(* IEC 61131-3 sources: NachHouse_CORE/V200/APP (part 6) *)

              47 : // HEV
						_Nh_POI_INI_NEW(cf:=xR^.h.cf.c, nd1:=xR^.h.cf.n, nd2:=xR^.h.cf.n, del:=true);
(*

             39 : // RFID card
                  _NhfVaz(pg := 133,  wh := 2, all := true);                   // vymaze vsetky vazby tohto oblubeneho ()
                  _NhDelRec(cf := xR^.h.cf.c, nd := xR^.h.cf.n);                  // vymaze zaznam
*)
//            ELSE
//                  xM^.wht  := 10;                                                                // nic sa nevymazalo, refresh dat od 1.riadku
//                  rmp      := 1;

             255 : // not acces right
		   			;
				END_CASE;
				IF rmp = 1 THEN
               _NhfVaz(vaz := 1, row := false, whf := 2, del := true, all := true);          // zoznam FAV, k HET ou
               _NhfVaz(vaz := 2, row := false, whf := 3, del := true, all := true);          // IO : in+ou WSB,TLA..PIR
               _NhfVaz(vaz := 3, row := false, whf := 3, del := true, all := true);          // IO : in+ou, vazby sCN
               _NhfVaz(vaz := 4, row := false, whf := 3, del := true, all := true);          // IO : in+ou, vazby ACT
            END_IF;
            IF xM^.wht = 0 THEN
               _NhxCfg(c := xR^.h.cf.c, n:= xR^.h.cf.n, x:=57);                                      // koli parametru
               IF xDev^.cf.par > 0 THEN
                  _NhFindDel(wh := 1, cx := aCfg[xR^.h.cf.c].par, nx := xDev^.cf.par, ok := false ); // vymazat parameter
               END_IF;
               _NhFindDel(wh := 0, cx := xR^.h.cf.c, nx := xR^.h.cf.n, ok := false );           // vymazat samotnu vetu aj jej pripadne parametre
               xM^.wht := 15;                                                                   // refresh pre vymazanu vetu
            END_IF;
            xM^.new     := 0;
            xA^.tch.cpy := 0;
            xA^.tch.del := 0;

     	103: // kopirovat VETU VAZBY a ZOSORTOVAT
            xM^.wht := 10;
            IF _NhfVaz(vaz := 2, whf := 10) THEN                                             // najde vetu vaz, ktora odpoveda riadku. AJ S PARAMTRAMI
               nd    := nDel+1;                                                              // nova veta by mala byt fyzicky za kopirovanou vetou
               yVaz  := xVaz^;                                                               // data kopirovanej vety
               yIO   := yVaz.ou;                                                             // zapamatanie zdroja DEV najma parametra
               nDel  := _NhFindDel(wh := 2, cx := 2, new := false, ok := false);             // skusi najst DEL-vetu vazby
               nDel  := _NhNewVaz(ok := nDel > 0, par := true, vaz := 2, nv := nDel);
               IF yIO.p > 0 AND yVaz.ou.p > 0  THEN
                  rb := _NhCpyRec(wh := 1,cf := aCfg[yIO.c].par ,ns := yIO.p, nd :=yVaz.ou.p);  // prekopiruje parameter
               END_IF;
               IF nDel > 0 THEN
                  _NhSrtVaz(vaz := 2, poz := nd, new := nDel);
//                  _NhSrtVaz(poz := nd, new := nDel);
                  xM^.wht  := 25;
               END_IF;
	            xM^.new     := 0;
   	         xA^.tch.cpy := 0;
      	      xA^.tch.del := 0;
            END_IF;

    	128: // oznacenie co kopirovat a kde
         _NhxPt(c := xR^.h.cf.c, n := xR^.h.cf.n, x:=33 );
			xRol := xPt;
			IF xU^.o[1].wh = 0 THEN 							// nemame zroj
				xU^.o[1].wh 	:= xR^.h.cf.n;             // vyberie sa zdroj
				xRol^.me.cpy 	:= 0;
			ELSIF xU^.o[1].wh = xR^.h.cf.n THEN       	// odznaci sa zdroj
				xU^.o[1].wh 	:= 0;
			ELSIF xRol^.me.cpy THEN
				xRol^.me.cpy 	:= 0;			              	// odznaci sa riadok
			ELSE
				xRol^.me.cpy 	:= 1;			          		// vyberie sa riadok ako ciel
			END_IF;

    	129: // zmena obrazka kopirovania v cat ROLETY + kopirovanie
			IF xA^.tch.obj = 2 THEN																	// START/Cancel
				xU^.o[1].wh := 0;
			END_IF;
			IF xU^.o[1].wh > 0 THEN                                              // mame cislo vety zdroja kopirovania
    			_NhxPt(c := 31, n := xU^.o[1].wh, x:=32 );
				xRol2 := xPt;
			END_IF;
			FOR nd := 1  TO aCfg[31].rec DO
				_NhxPt(c := 31, n := nd, x:=31 );
				xRol 				:= xPt;
				IF xU^.o[1].fn = 44 AND xRol^.me.cpy AND xU^.o[1].wh > 0 THEN     // mame zdroj aj tato veta je oznacena
					xRol^.cx.cf := xRol2^.cx.cf;												// prekopiruje zo zdroja
				END_IF;
				xRol^.me.cpy 	:= 0; 															// vymaze ciel kopirovania
  			END_FOR;
//			xU^.o[1].wh 		:= 0;

			IF xU^.o[2].fn  = 45 THEN														// sivy COPY vpravo
				// prepnute na kopirovanie
				xU^.o[2].fn  :=  46;				 	                              	// cancel vpravo
				xU^.o[1].fn  :=  44;																// zlty copy vlavo
				xU^.o[1].cm  := 129;
			ELSE
				// default
				xU^.o[2].fn  :=  45;
				xU^.o[1].fn  :=  0;
				xU^.o[1].cm  :=  0;
				_Nh_Brw_Dsh_Chg();																// nastavi ikonu kopirovania
			END_IF;

    	130: // kopirovanie POI pre typove dni {predtym 45}
				_Nh_xPod_Map(cf:=xF^.cf.c, nd:=xF^.cf.n, WhtPoi:=xM^.pod.po.WhtPoi);
				xPod2 := xPod;															// zdroj dni kopirovania

				IF xM^.pod.cp.all  THEN
            	FOR nd := 1 TO aCfg[xF^.cf.c].rec DO
						IF _NhxPt(c:=xF^.cf.c, n:=nd, x:=130) AND nd <> xF^.cf.n AND xPt^.ok.cpy THEN	// prechadza DEV kam sa ma kopirovat (ROM/HET/VEN..., vyluci zdroj
							xPt^.ok.cpy := false;                                       // odznaci priznak kopirovania
							_Nh_xPod_Map(cf:=xF^.cf.c, WhtPoi:=xM^.pod.po.WhtPoi);											// ciel namapuje dni xPod podla druhu CF
							FOR i := 1 TO 11 DO
		                  IF xM^.pod.cp.dst[i] AND xPod2^.poi[ i ] > 0 THEN			// den v zdroji sa kopiruje a ma vetu POI
	   	         			IF _NhxPt(c := 26, n := xPod2^.poi[ i ],x:=26) THEN
					   				xPox  	:= xPt;												// zdrojova veta POI
										IF xPod^.poi[ i ] > 0 THEN									// ciel ma vetu POI
			   	         			IF _NhxPt(c := 26, n := xPod^.poi[ i ],x:=26) THEN
							   				xPox2  	:= xPt;										// cielova veta POI
      										xPox2^	:= xPox^;                           // prepise ciel zdrojom
      									END_IF;
										END_IF;
									END_IF;
								END_IF;
	                  END_FOR;
						END_IF;
					END_FOR;
//					_NhDevSetCpy(set:=false, cf:=xF^.cf.c, nd:=1, rec:=aCfg[xF^.cf.c].rec);
		         _NheLvl(lvl:=-2);                                              // o LVL dopredu

				ELSIF xPod2^.poi[ xM^.pod.cp.src ] > 0 THEN                                // mame zdroj > 0
	            IF _NhxPt(c := 26, n := xPod2^.poi[ xM^.pod.cp.src ],x:=25) THEN  	// najde zdroj
	   				xPox  := xPt;																	// zdrojova veta POI
						FOR i := 1 TO 11 DO
	                  IF xM^.pod.cp.dst[i] AND xPod2^.poi[ i ] > 0 THEN				// do ciela sa kopiruje a ciel ma vetu POI
	            			IF _NhxPt(c := 26, n := xPod2^.poi[ i ],x:=26) THEN  		// cielova veta POI
				   				xPox2  	:= xPt;													// cielova veta POI
									xPox2^	:= xPox^;                                    // prepise ciel zdrojom
								END_IF;
							END_IF;
                  END_FOR;
   				END_IF;
				END_IF;
				_NheBrw(wht:=12);

    	131: // kopirovanie celych ROM + oznacenie kopirovanie
			_NheBrw(wht:=12);
         xU^.o[2].cm := 131;
    		CASE xU^.o[2].fn OF
			 	45: 	// sive copy
						xU^.o[2].fn := 44;														// zlte copy
						xM^.pod.cp.all	:= 1;
						FOR i := 1 TO 11 DO
							xM^.pod.cp.dst[i] := 1;
                  END_FOR;
			 	44: 	// zlte copy
						xU^.o[2].fn := 45;														// zlte copy
						xM^.pod.cp.all	:= 0;

				ELSE  xU^.o[2].fn := xU^.o[2].wh;
						xM^.pod.cp.all	:= 0;
						xM^.pod.cp.cpy	:= 0;
			END_CASE;
			xA^.tch.obj	:= -1;										// zaisti aby sa objekt nevybral , inak by sa zobrazovalo to co je xU^.o[2].wht
			xA^.tch.cmd := 207;										// urobi refresh uz nadefinovaneho screenu

    	132: // browser - vyber kopirovania
         IF _NheLvl( lvl := 4) THEN
            _Nh_Web_CMD_Screen(obj := 60);
				_NhDevSetCpy(set:=false, cf:=xF^.cf.c, nd:=1, rec:=aCfg[xF^.cf.c].rec);		// resetne priznak cpy
         END_IF;
    	133: // oznacenie - kopirovania
			IF xA^.tch.mnu AND xA^.tch.obj = 2 THEN												// oznacit vsetko
				_NhDevSetCpy(set:=NOT xM^.pod.cp.chk, cf:=xF^.cf.c, nd:=1, rec:=aCfg[xF^.cf.c].rec);
				xM^.pod.cp.chk := NOT xM^.pod.cp.chk;
			ELSIF xA^.tch.row >= 0 THEN
				IF xF^.cf.n <> xB^.r[xA^.tch.row].h.cf.n THEN										// dotyk nad inym ako zdrojom
					_NhDevSetCpy(set:=NOT xPt^.ok.cpy, cf:=xB^.r[xA^.tch.row].h.cf.c, nd:=xB^.r[xA^.tch.row].h.cf.n, rec:=xB^.r[xA^.tch.row].h.cf.n);
					xM^.pod.cp.chk := _NhDevSetCpy(chk:=true, set:=NOT xM^.pod.cp.chk, cf:=xF^.cf.c, nd:=1, rec:=aCfg[xF^.cf.c].rec);
				END_IF;
			END_IF;
			xA^.tch.mnu	:= 0;
//			xU^.o[1].fn := _Nh_O12(xM^.pod.cp.chk,44,45);
			xU^.o[1].fn := _Nh_O12(xM^.pod.cp.chk,44,6);

    	136: // <  O UROVEN SPAT z REGulatora
         _NhxPt(c := xF^.cf.c, n := xF^.cf.n, x:=136 );                     // xDev,xCfg,xPar pre aktualny riadok
			xHet := xPt;
			xHet^.cx.reg.ModeFromSrc := true;
         _NheLvl(lvl:=-1);                                              // o LVL dopredu
         xM^.htt :=  '';

		137: // prepnut MAN/AUTO
      	   xDev^.al.in.cmd := 37;
    	138: // nastav MAN
   	      xDev^.al.in.cmd := 38;
    	139: // nastav AUTO
	         xDev^.al.in.cmd := 39;
    	140: // nastavit wRGBo na TGL
      	   _NhxDev(c := xF^.cf.c, n := xF^.cf.n, x:=36 );                     // xDev,xCfg,xPar pre aktualny riadok
   	      xDev^.al.in.cmd := 36;
    	141: // vyrobit HET
				aSys.ini := 11;
				RETURN;

    	190: // roleta - vyber hore / dolu
         _NhxDev2(c := xR^.h.cf.c, n := xR^.h.cf.n, x:=35 );                     // xDev,xCfg,xPar pre aktualny riadok
         ok := false;
         FOR j := 1 TO 10 DO
            IF ok THEN
               xR^.o.ob[j].btn := false;
            ELSIF xA^.tch.obj = j THEN
//               xDev2^.al.in.cmd := 239+SINT_TO_USINT(j);                // cislo cmd od 240...249
//               xR^.o.ob[j].btn := NOT xR^.o.ob[j].btn;

               IF xR^.o.ob[j].btn=false THEN                               // teraz je este vypnuty, ale bude zapnuty btn v pocedure show...
                  xDev2^.al.in.cmd := 239+SINT_TO_USINT(j);                // cislo cmd od 240...249
               ELSE                                                        // bude vypnuty
                  xDev2^.al.in.cmd := 255;                                 // stop vsetkemu co bezi
               END_IF;
               ok := true;
            END_IF;
         END_FOR;

         xM^.wht := -1;                                     // len cisty refresh existujucich dat v riadku bez predefinovania dat

(*
    191: // roleta setup : prepnut HORE/DOLU
         _NhxDev2(c := xR^.h.cf.c, n := xR^.h.cf.n, x:=36 );                     // xDev,xCfg,xPar pre aktualny riadok
         xRol := xDev2;
         CASE xA^.tch.obj OF
           7 : xRol^.al.Qf := 1; xRol^.al.Qx := 0;
           8 : xRol^.al.Qf := 0; xRol^.al.Qx := 1;
         END_CASE;
         xM^.wht     := 30;
*)

    	199: // DOTYK NAD IKONOU Day Of Week
         IF _NheLvl( lvl := 1 ) THEN                                 // nadefinuje menu stanky
            xL^.obj        := 200;                                      // podhodi sa 200
            xA^.tch.obj    := 3;                                        // prvy objekt = 3
            xF^.rom        := 199;                                      // podla tohto sa nadefinuje menu
            xA^.tch.cm     := 200;
            xA^.tch.cmd    := 200;                                      // vrati sa uz do 200
            RETURN;
         END_IF;

    	200: // DOTYK NAD HLAVNYM OBRAZOK RIADKA = VLASTNOSTI
         xM^.wht     := -1;
         IF xL^.obj = 200 THEN                                           // stranka uz je, zmenilo sa nieco v menu
            xU^.n    := SINT_TO_USINT(xA^.tch.obj);                        // nastavi sa stranka odpovedajuca obj
            xM^.wht  := 20;                                             // predefinuju sa objekty
            yIO      := xB^.r[0].h.cf;

         ELSIF _NheLvl( lvl := 1 ) THEN                                 // nadefinuje menu stanky
            xL^.obj     := 200;
            xM^.wht     := 20;

(*
            IF xR^.h.chk AND xA^.tch.obj = 4 THEN //AND xR^.o.ob[4].cf.c > 0 THEN // v objekte 4 je vaba so spravnym parametrom
               xF^.cf  := xR^.o.ob[4].cf;                             // hlavicka sa preberie z riadka
            END_IF;
*)

         END_IF;

    	201: // nadefinovat LOKALNU,externu stranku
            IF xL^.obj  = 201 THEN
               _NhxDev2(c := xF^.cf.c, n := xF^.cf.n, x:=61);
               xUsr2       := xDev2;
              IF xM^.htx = 10 THEN //; xM^.htt = 'USR_NHF.XML' THEN
                  xM^.htx     := 11;
                  xM^.htt     := 'US2_NHF.XML';
                  xU^.o[2].fn := 0;                                             // vsetky rom
                  xU^.o[2].cm := 0;                                             // vsetky rom
                  xU^.o[1].cm := 201;                                             // vsetky rom
						IF xUsr^.ok.ref THEN
	                  xUsr2^      := yUSR;
						END_IF;
               ELSIF xM^.htx = 11   THEN  //;xM^.htt = 'US2_NHF.XML' THEN
                  xM^.htx     := 10;
                  xM^.htt     := 'USR_NHF.XML';
                  xU^.o[2].fn := 7;                                             // vsetky rom
                  xU^.o[2].cm := 201;                                             // vsetky rom
                  xU^.o[1].cm := 202;                                             // vsetky rom
						IF xUsr^.ok.ref THEN
	                  xUsr2^      := yUSR;
						END_IF;
               END_IF;
					xUsr^.ok.ref := false;

            ELSIF _NheLvl( lvl := 1 ) THEN                                 // nadefinuje menu stanky
               xL^.obj     := 201;
               _NhxDev2(c := xR^.h.cf.c, n := xR^.h.cf.n, x:=68);
               xUsr2       	:= xDev2;
					xUsr^.ok.ref	:= false;
               CASE xR^.h.cf.c OF
                 22: // USRs;
							yUsr        := xUsr2^;
                     IF  xA^.usr = 1 OR xA^.UsrRight >=2 THEN       							// moze lne spravca a admin
                        xM^.htx     := 10;
                        xM^.htt     := 'USR_NHF.XML';
                        xU^.o[2].fn := 7;                                             // vsetky rom
                        xU^.o[2].cm := 201;                                             // vsetky rom
                     ELSE
                        _NheLvl( lvl := -1 );
                     END_IF;
               ELSE
                    	_NheLvl( lvl := -1 );
                     RETURN;
               END_CASE;
               xU^.o[1].cm := 202;                                             // vsetky rom
               xM^.frm     := true;
            END_IF;
            xM^.wht := -1;

    	202: // ukoncit-ulozit data lokalnej stranky
            _NhWebSave();

    	203: // VSTUP DO SUB-MENU FRAME
 				_Nh_FRM_Read(frm:=USINT_TO_UINT(xU^.o[ xA^.tch.obj ].frm)); 	// v tom istom LVL nacita ine menu vo FRM
				xA^.tch.obj := USINT_TO_SINT(xU^.n);
      	   xA^.tch.cmd    := 206;                                      // vrati sa uz do 200

    	204: // VSTUP DO MENU FRAME
         IF _NheLvl( lvl := 1 ) THEN                                 // nadefinuje menu stanky
            xL^.vaz     := xM^.lvd[xM^.lvl-1].vaz;
            xL^.chk     := xM^.lvd[xM^.lvl-1].chk;
            xL^.rw1     := xM^.lvd[xM^.lvl-1].fil.cf;       // hlavicku browsu, kde bola veta z ktorej sa islo
            xB^.r[0]    := xR^;                             // v r[0] bude cela veta a odial r[0].h.chk - ci bola vazba
            xL^.obj     := 205;
         END_IF;
    	205: // ZMENA MENU VO FRAME

	 	210: // DOTYK Weather
         IF _NheLvl( lvl := 3) THEN
				xF^.cf.c			:= 3;
				xF^.cf.n			:= 1;
	   	   _Nh_Lang(id := 354 ,txt := ADR( xL^.naz ),zn:=20);
				_Nh_FRM_Read(frm:=68);
   	      xL^.obj        := 205;                                      // podhodi sa 200
      	   xA^.tch.cmd    := 206;                                      // vrati sa uz do 200
         END_IF;

		215: // DOTYK HOME-typove dni
         IF _NheLvl( lvl := 3) THEN
				xF^.cf.c			:= 3;
				xF^.cf.n			:= 1;
            _NhxPt(c := xF^.cf.c, n := xF^.cf.n, x:=7);                               // nazov DEV
            xL^.naz := xPt^.cf.Name;
				_Nh_FRM_Read(frm:=75);
   	      xL^.obj        := 205;                                      // podhodi sa 200
      	   xA^.tch.cmd    := 206;                                      // vrati sa uz do 200
         END_IF;

   { $IFDEF __NH_DALI }

    	247: // funkcie brw-DALI-SLAVE-zmena v spodnom menu - rozne filtre, akcie na BTN
         xM^.wht := 20;
         IF xF^.cf.c = 42 THEN                                     // spodne menu pre browser DLS/DLg - v hlavicke je master
            _Nh_Chk_DALI(set:=true, mnu:=xA^.tch.obj);
            xU^.n := 0;
         ELSIF xR^.h.cf.c = 42 THEN                               // riadok je DLM - akcia od btn
            xM^.wht  := -1;                                        // v tomto cykle sa nepokracuje do browsu, lebo sa nastavuje DEV , az v druhom cykle
            xDLm     := xDev;
            ii       := INT_TO_USINT(xR^.h.cf.n);
            xDlfb    := ADR(aDali[ii]);
            CASE xA^.tch.obj OF
              2 : // ON/OFF - master
                  IF xDLfb^.cmd[1].cmd > 0 THEN                                                   // ak prebieha nejaku task, breakne ho
//                     IF xDlfb^.cmd[1].Break THEN                          // bezi proces, ktory sa neda braknut                                 // ak prebieha nejaku task, breakne ho
//                        xDLfb^.Break := true;
//                     END_IF;
                  ELSE
                     xDev^.al.in.cmd   := 1;                      // prepni bez oneskorenia
                     xDev^.al.in.par   := 0;                      // pri takomto zadani sa zoberie default parameter
                     xM^.wht           := 0;                      // v tomto cykle sa nepokracuje do browsu, lebo sa nastavuje DEV , az v druhom cykle
                  END_IF;
              4 : // vstup do brw-DLs z mastra
                  IF _NheLvl( lvl := 1) THEN                      // o LVL dopredu bez prebratia menu
                     _Nh_Web_CMD_Screen(obj := 48);
                  END_IF;
              6 : // vstup do brw-DLg z mastra
                  IF _NheLvl( lvl := 1) THEN                      // o LVL dopredu bez prebratia menu
                     _Nh_Web_CMD_Screen(obj := 47);                        // VAZBY,LIST....
                  END_IF;

            END_CASE;
         END_IF;

    	249: // DALI- browser MASER + SLAVE
            xM^.wht        := -1;
            IF xA^.tch.Q THEN
               j  := xA^.tch.obj;
               xO := ADR(xR^.o.ob[j]);
            END_IF;
            CASE xR^.h.cf.c OF
            42:   // master
                  xDLm     := xDev;
                  ii       := INT_TO_USINT(xR^.h.cf.n);
                  xDlfb    := ADR(aDali[ii]);
                  CASE xA^.tch.obj OF
                     2: // ON/OFF
                        xDev^.al.in.cmd   := 1;                                     // prepni bez oneskorenia
                        xDev^.al.in.par   := 0;                                     // pri takomto zadani sa zoberie default parameter
                        xM^.wht           := 0;                                        // v tomto cykle sa nepokracuje do browsu, lebo sa nastavuje DEV , az v druhom cykle
                     4 : // brows Sha
                        IF _NheLvl( lvl := 1) THEN                      // o LVL dopredu bez prebratia menu
                           _Nh_Web_CMD_Screen(obj := 48);                        // VAZBY,LIST....
                        END_IF;
                  END_CASE;
            43:   // slave
                  xDLs  	:= xDev;
		            dlsl     := _Nh_DL_sha(nd := xR^.h.cf.n);
   		         dlma     := _Nh_DL_sha(ma := true, nd := xR^.h.cf.n);

                  CASE xA^.tch.obj OF
                     1: // hlavna ikona = frame
                        IF _NheLvl( lvl := 1 ) THEN                                 // nadefinuje menu stanky
                           xL^.obj     := 205;
                        END_IF;
                     6 : // priradit DLs->DLs
                        IF _NheLvl( lvl := 1) THEN
                           _Nh_Web_CMD_Screen(obj := 47);
                        END_IF;
                     2: // ON/OFF len pre Miboxer z 1 adresou a RGBW

                        xDev^.al.in.cmd   := 43;                                     // prepni bez oneskorenia
                        xDev^.al.in.par   := 0;                                     // pri takomto zadani sa zoberie default parameter
                        xM^.wht           := 0;                                        // v tomto cykle sa nepokracuje do browsu, lebo sa nastavuje DEV , az v druhom cykle

                  END_CASE;
            ELSE
            ;
            END_CASE;

   { $END_IF }

    	250: //   prepinanie rezimu setup
            _NhDefSet(chg := true);
            xM^.wht     := -1;

    	251: // dotyk/podrzanie na SLIDER
            xM^.wht := -1;                                     // len cisty refresh existujucich dat v riadku bez predefinovania dat
    	252: // // vypis od 1.riadka s predefinovanim dat v riadku
            xM^.wht := 10;                                     //***---*** POZOR !!! zmena - dotyk sa presuva do objektu spat
    	253: // len pre predefinovanie objektov v NhBrw200
            xM^.wht := 30;
    	254: // kompletny refresh browsu s novym indexom a datami od existujuceho 1.riadka
            xM^.wht := 25;
    	255: // nic sa nedeje, riadi si to
         ;
//         aSys.RestDev := true;
   END_CASE;

   IF aWht.n < 6 THEN
      xA^.tch.wht := xM^.wht;
      aWht.t[aWht.n] := xA^.tch;
      aWht.t[aWht.n].cmdNext := cmd;
      aWht.t[aWht.n].xMwht  := xM^.wht;
      aWht.n := aWht.n + 1;
   END_IF;

   IF xL^.obj = 205   THEN
      IF _Nh_Shw_FRM() = false THEN
         RETURN;
      END_IF;
   ELSIF xM^.wht = 0 THEN                                            // neprekreslule sa brows
      ;
   ELSIF xM^.delay > 0 THEN                                       // cakanie na delay
      xM^.delay := xM^.delay - MIN(xM^.delay, aSys.mSec);
      RETURN;
   ELSIF xL^.obj = 0 THEN                                          // HOME screen
      IF _Nh_Frm_HOM() = false THEN
         RETURN;
		END_IF;
(*
   ELSIF xL^.obj = 200 THEN                                           // PARAMETERS
      IF _NhBrw200() = false THEN
         RETURN;
      END_IF;
*)
   ELSIF _Nh_Web_BRW() = false THEN                              // ZAKLADNY 6-riadkovy BROWSER
      RETURN;
   END_IF;

   xM^.wht     := 0;
   xA^.tch.cmd := cmd;
   xM^.delay   := delay;

END_FUNCTION

{ $ END_IF }

(* ---- _Nh_WRK.st ---- *)
{ $IFDEF __NH_WRK }

VAR_GLOBAL                                            // len pre ladenie
   _NhWrk      {HIDDEN} : BOOL := true ;
   { $ IF CPU_CODE > 1999  }
   yIdx         : ARRAY[1..30]	OF NH_IDX;

	yScn			{HIDDEN} : ARRAY[1..50]  OF NH_SCN;
   ypScn 		{HIDDEN} : ARRAY[1..20]  OF NH_SVA_PAR;
	yAct			{HIDDEN} : ARRAY[1..50]  OF NH_ACT;
//	yAla			{HIDDEN} : ARRAY[1..10]  OF NH_ALA;

//		yyVaz	{HIDDEN}	: ARRAY[1.._Nh_VAZ] OF NH_VAZ_CFG ;

		yVaz1			{HIDDEN} : ARRAY[1..50]  OF NH_VAZ;
//	  	yVaz2 		{HIDDEN} : ARRAY[1..150] OF NH_VAZ;
//		yVaz3			{HIDDEN} : ARRAY[1..50]  OF NH_VAZ;
//   	yVaz4			{HIDDEN} : ARRAY[1..80]  OF NH_VAZ;

//  		yGlb			{HIDDEN} : ARRAY[1..1]   OF NH_GLB;
	   yRom			{HIDDEN} : ARRAY[1..30]	OF NH_ROM;
   	yZon			{HIDDEN} : ARRAY[1..10]	OF NH_ROM;
	   ypZon 		{HIDDEN} : ARRAY[1..20]  OF NH_ZON_PAR;
   	yRoW        {HIDDEN} : ARRAY[1..10]  OF NH_WRK_ROM;
		yZoW        {HIDDEN} : ARRAY[1.. 7]  OF NH_WRK_ROM;
		yRol			{HIDDEN} : ARRAY[1..20]  OF NH_ROL;
   	ypRol 		{HIDDEN} : ARRAY[1..100]  OF NH_ROL_PAR;       // 12
//   	yPoi			{HIDDEN} : ARRAY[1..50]  OF NH_POI;

		yTgl			{HIDDEN} : ARRAY[1..30]  OF NH_TGL;
  		ypTgl 		{HIDDEN} : ARRAY[1..120]  OF NH_WSB_PAR;

   ySvd 			{HIDDEN} : ARRAY[1..10]  OF NH_SVD;
   pSvd 			{HIDDEN} : ARRAY[1..100]  OF NH_SVD_PAR;
  	ySva 			{HIDDEN} : ARRAY[1..10]  OF NH_SVA;  //10
  	pSva 			{HIDDEN} : ARRAY[1..40]  OF NH_SVA_PAR;
   yRgb 			{HIDDEN} : ARRAY[1..10]  OF NH_RGB;
	yyRgb 			{HIDDEN} : NH_RGB;
   pRgb 			{HIDDEN} : ARRAY[1..20]  OF NH_RGB_PAR;

	yTve			{HIDDEN} : ARRAY[1..20]  OF NH_TVE;
//	yHet			{HIDDEN} : ARRAY[1..10]  OF NH_HET;  // 20
(*

 	ypHet 		{HIDDEN} : ARRAY[1..20]  OF NH_HET_PAR;       // 10

//	yHev			{HIDDEN} : ARRAY[1..5]   OF NH_HET;  // 20

	yVen 			{HIDDEN} : ARRAY[1..10]  OF NH_TVE;
*)

(*
		yLux			{HIDDEN} : ARRAY[1..5]  OF NH_LUX;
   	yTer 			{HIDDEN} : ARRAY[1..40]  OF NH_TER;
	   yTeh 			{HIDDEN} : ARRAY[1.. 5]  OF NH_TER;
   	yTek 			{HIDDEN} : ARRAY[1.. 5]  OF NH_TER;

*)
//		yRhx			{HIDDEN} : ARRAY[1..2]  OF NH_LUX;
//	yCer			{HIDDEN} : ARRAY[1..3]	 OF NH_TVE;
//	yKot			{HIDDEN} : ARRAY[1..5]	 OF NH_TVE;
//  	yTim			{HIDDEN} : ARRAY[1..10]  OF NH_TIM;
//	yKey			{HIDDEN} : ARRAY[1..3]   OF NH_KEY;

(*
	yDls			{HIDDEN} : ARRAY[1..130]   OF NH_DLS;
	pDls			{HIDDEN} : ARRAY[1..200]   OF NH_RGB_PAR;
	yDlm			{HIDDEN} : ARRAY[1..4]   OF NH_DLM;
	yDlg			{HIDDEN} : ARRAY[1..32]   OF NH_DLG;
*)

//    	yMsg			{HIDDEN} : ARRAY[1..3] OF NH_MSG;

//	  yCat			{HIDDEN} : ARRAY[1..70]	OF NH_CAT;

      yVvo 			{HIDDEN} : ARRAY[1..4]   OF NH_VVO;

   yWsb 			{HIDDEN} : ARRAY[1..30]  OF NH_WSB;
   ypWsb 		{HIDDEN} : ARRAY[1..50]  OF NH_WSB_PAR;

   yTla 			{HIDDEN} : ARRAY[1..10]  OF NH_TLA;

//   ytGl		 {HIDDEN} : ARRAY[1..10]  OF NH_TGL;
//	yPIR			{HIDDEN} : ARRAY[1..50]  OF NH_PIR;
//   ypPir 		{HIDDEN} : ARRAY[1..10]  OF NH_PIR_PAR;

//	yCox			{HIDDEN} : ARRAY[1..10]  OF NH_LUX;

//	yDor			{HIDDEN} : ARRAY[1..10]  OF NH_DOR;

//	yFav			{HIDDEN} : ARRAY[1..10]  OF NH_FAV;
//   yZas 			{HIDDEN} : ARRAY[1..15]  OF NH_SVD;
//   pZas 			{HIDDEN} : ARRAY[1..10]  OF NH_SVD_PAR;
//	yyUsr			{HIDDEN} : ARRAY[1..7]   OF NH_USR;

//	ySmw			{HIDDEN} : ARRAY[1..10]  OF NH_SMW;

//	yGat			{HIDDEN} : ARRAY[1.. 5]  OF NH_GAT;
//	yBra			{HIDDEN} : ARRAY[1.. 5]  OF NH_GAT;
//   ypGat 		{HIDDEN} : ARRAY[1..10]  OF NH_GAT_PAR;       // 13

//	ySir			{HIDDEN} : ARRAY[1.. 5]  OF NH_SVD;
//	yBlk			{HIDDEN} : ARRAY[1.. 5]  OF NH_BLK;
//	yBlx			{HIDDEN} : ARRAY[1.. 5]  OF NH_BLX;
//	yBtn			{HIDDEN} : ARRAY[1..20]  OF NH_BTN;
(*
//	yAcl			{HIDDEN} : ARRAY[1..20]  OF NH_VAZ;
*)
//	yVcf			{HIDDEN} : ARRAY[1..150]  OF NH_VAZ_VCF;
//	ySbj			{HIDDEN} : ARRAY[1..4]  OF NH_SBJ;

   { $ ELSE  }

//   	yPoi			{HIDDEN} : ARRAY[1..20]  OF NH_POI;
//	   yRom			{HIDDEN} : ARRAY[1..10]	    OF NH_ROM;
//   	yZon			{HIDDEN} : ARRAY[1..10]	  OF NH_ROM;
//    yRoW        {HIDDEN} : ARRAY[1..10]    OF NH_WRK_ROM;
   { $ END_IF  }

END_VAR

	FUNCTION	_DevDataX {HIDDEN} : BOOL
      VAR_IN_OUT
         aNh   : NH_CFG_CFG;
         dst   : USINT;
      END_VAR
      VAR_INPUT
         n    : UDINT := 10;
      END_VAR
      memsetEx(val := 0,length := n * aNh.Siz , dest := dst ); // vycisti
      IF aNh.Ram > 0 THEN
         MemcpyEx(length := Min(n, INT_TO_UDINT(aNh.Rec)) * aNh.Siz , source := void( mRam[ aNh.Ram ]), dest := dst);
      END_IF;
      _DevDataX := true;
   END_FUNCTION

   FUNCTION	_NhDataWrk {HIDDEN} : BOOL
      VAR_INPUT
         Yes  : BOOL := true ;
      END_VAR
      IF Yes = false THEN
         RETURN;
      END_IF;
		_NhDataWrk :=  TRUE;
      { $ IF CPU_CODE > 1999  }
         { $IFDEF yGlb }
            _DevDataX(aNh := VOID(aCfg[25]), dst := VOID(yGlb), n :=1);
         { $END_IF }
         { $IFDEF yRom }
            _DevDataX(aNh := VOID(aCfg[ 1]), dst := VOID(yrom), n :=30);
         { $END_IF }
         { $IFDEF yPoi }
            _DevDataX(aNh := VOID(aCfg[26]), dst := VOID(yPoi), n := 50);
         { $END_IF }
      { $ ELSE  }
         { $IFDEF yRom }
            _DevDataX(aNh := VOID(aCfg[ 1]), dst := VOID(yrom), n :=10);
         { $END_IF }
         { $IFDEF yPoi }
            _DevDataX(aNh := VOID(aCfg[26]), dst := VOID(yPoi), n := 20);
         { $END_IF }
      { $ END_IF  }

      { $IFDEF yMsg }
      _DevDataX(aNh := VOID(aCfg[46]), dst := VOID(yMsg), n :=3);
      { $END_IF }

      { $IFDEF ycat }
      _DevDataX(aNh := VOID(aCfg[ 2]), dst := VOID(yCat), n :=70);
      { $END_IF }
      { $IFDEF yZon }
      _DevDataX(aNh := VOID(aCfg[ 3]), dst := VOID(yZon), n :=10);
      { $END_IF }
      { $IFDEF ypZon }
      _DevDataX(aNh := VOID(aPar[5]), dst := VOID(ypZon), n :=20);
      { $END_IF }
      { $IFDEF yHet }
      _DevDataX(aNh := VOID(aCfg[ 6]), dst := VOID(yHet));
      { $END_IF }
      { $IFDEF yHev }
      _DevDataX(aNh := VOID(aCfg[47]), dst := VOID(yHev), n:=5);
      { $END_IF }
      { $IFDEF yKot }
      _DevDataX(aNh := VOID(aCfg[ 7]), dst := VOID(yKot), n:=5);
      { $END_IF }
      { $IFDEF ytve }
      _DevDataX(aNh := VOID(aCfg[ 8]), dst := VOID(yTve), n:=20);
      { $END_IF }
      { $IFDEF ycer }
      _DevDataX(aNh := VOID(aCfg[ 9]), dst := VOID(yCer), n := 3);
      { $END_IF }
      { $IFDEF ysvd }
      _DevDataX(aNh := VOID(aCfg[10]), dst := VOID(ySvd));
      { $END_IF }
      { $IFDEF ySva }
      _DevDataX(aNh := VOID(aCfg[11]), dst := VOID(ySva));
      { $END_IF }
      { $IFDEF yVvo }
      _DevDataX(aNh := VOID(aCfg[49]), dst := VOID(yVvo), n :=4);
      { $END_IF }
      { $IFDEF yRgb }
      _DevDataX(aNh := VOID(aCfg[12]), dst := VOID(yRgb));
      { $END_IF }
      { $IFDEF ywsb }
      _DevDataX(aNh := VOID(aCfg[13]), dst := VOID(yWsb), n :=30);
      { $END_IF }
      { $IFDEF ytla }
      _DevDataX(aNh := VOID(aCfg[14]), dst := VOID(yTla));
      { $END_IF }
      { $IFDEF ypir }
      _DevDataX(aNh := VOID(aCfg[15]), dst := VOID(yPir), n :=50);
      { $END_IF }
      { $IFDEF yter }
      _DevDataX(aNh := VOID(aCfg[16]), dst := VOID(yTer), n :=40);
      { $END_IF }
      { $IFDEF yteh }
      _DevDataX(aNh := VOID(aCfg[17]), dst := VOID(yTeh), n := 5);
      { $END_IF }
      { $IFDEF ytek }
      _DevDataX(aNh := VOID(aCfg[18]), dst := VOID(yTek), n := 5);
      { $END_IF }
      { $IFDEF ylux }
      _DevDataX(aNh := VOID(aCfg[19]), dst := VOID(yLux), n := 5);
      { $END_IF }
      { $IFDEF yRhx }
      _DevDataX(aNh := VOID(aCfg[51]), dst := VOID(yRhx), n := 2);
      { $END_IF }
      { $IFDEF yfav }
      _DevDataX(aNh := VOID(aCfg[20]), dst := VOID(yFav));
      { $END_IF }
      { $IFDEF yzas }
      _DevDataX(aNh := VOID(aCfg[21]), dst := VOID(yZas), n:=15);
      { $END_IF }
      { $IFDEF yDor }
      _DevDataX(aNh := VOID(aCfg[33]), dst := VOID(yDor));
      { $END_IF }
      { $IFDEF yyUsr }
      _DevDataX(aNh := VOID(aCfg[22]), dst := VOID(yyUsr), n:=7);
      { $END_IF }
      { $IFDEF yven }
      _DevDataX(aNh := VOID(aCfg[23]), dst := VOID(yVen));
      { $END_IF }
      { $IFDEF yKey }
      _DevDataX(aNh := VOID(aCfg[24]), dst := VOID(yKey), n := 3);
      { $END_IF }
      { $IFDEF ysmw }
      _DevDataX(aNh := VOID(aCfg[45]), dst := VOID(ySmw));
      { $END_IF }
      { $IFDEF yRol }
      _DevDataX(aNh := VOID(aCfg[31]), dst := VOID(yRol), n:=20);                    //ROL
      { $END_IF }
      { $IFDEF yBra }
      _DevDataX(aNh := VOID(aCfg[37]), dst := VOID(yBra), n := 5);            //BRA - stara
      { $END_IF }
      { $IFDEF yGat }
      _DevDataX(aNh := VOID(aCfg[37]), dst := VOID(yGat), n := 5);            //BRA
      { $END_IF }
      { $IFDEF ySir }
      _DevDataX(aNh := VOID(aCfg[32]), dst := VOID(ySir), n := 5);            //SIR
      { $END_IF }
      { $IFDEF yBlk }
      _DevDataX(aNh := VOID(aCfg[35]), dst := VOID(yBlk), n := 5);            //BLK
      { $END_IF }
      { $IFDEF yBlx }
      _DevDataX(aNh := VOID(aCfg[36]), dst := VOID(yBlX), n := 5);            //BLK
      { $END_IF }
      { $IFDEF yTgl }
      _DevDataX(aNh := VOID(aCfg[40]), dst := VOID(yTgl), n :=30);
      { $END_IF }
      { $IFDEF yBtn }
      _DevDataX(aNh := VOID(aCfg[41]), dst := VOID(yBtn), n := 20);
      { $END_IF }
      { $IFDEF yDlm }
      _DevDataX(aNh := VOID(aCfg[42]), dst := VOID(yDlm), n := 4);
      { $END_IF }
      { $IFDEF yDls }
      _DevDataX(aNh := VOID(aCfg[43]), dst := VOID(yDls), n := 130);
      { $END_IF }
      { $IFDEF yDlg }
      _DevDataX(aNh := VOID(aCfg[44]), dst := VOID(yDlg), n := 32);
      { $END_IF }
      { $IFDEF yTim }
      _DevDataX(aNh := VOID(aCfg[50]), dst := VOID(yTim), n := 10);
      { $END_IF }
      { $IFDEF yScn }
      _DevDataX(aNh := VOID(aCfg[ 4]), dst := VOID(yScn), n := 50);
      { $END_IF }
      { $IFDEF yact }
      _DevDataX(aNh := VOID(aCfg[ 5]), dst := VOID(yAct), n:= 50);
      { $END_IF }
      { $IFDEF yAla }
      _DevDataX(aNh := VOID(aCfg[48]), dst := VOID(yAla));
      { $END_IF }
      { $IFDEF yVaz1 }
      _DevDataX(aNh := VOID(aVaz[ 1]), dst := VOID(yVaz1), n := 50);
      { $END_IF }
      { $IFDEF yVaz2 }
      _DevDataX(aNh := VOID(aVaz[ 2]), dst := VOID(yVaz2), n :=150);
      { $END_IF }
      { $IFDEF yVaz3 }
      _DevDataX(aNh := VOID(aVaz[ 3]), dst := VOID(yVaz3), n := 50);
      { $END_IF }
      { $IFDEF yVaz4 }
      _DevDataX(aNh := VOID(aVaz[ 4]), dst := VOID(yVaz4), n :=80);
      { $END_IF }

(*
      { $IFDEF yAcl }
      _DevDataX(aNh := VOID(aVaz[ 5]), dst := VOID(yAcl), n := 20);
      { $END_IF }
*)

      { $IFDEF pSvd }
       _DevDataX(aNh := VOID(aPar[1]), dst := VOID(pSvd), n := 100);
      { $END_IF }
      { $IFDEF pSva }
      _DevDataX(aNh := VOID(aPar[2]), dst := VOID(pSva), n := 40);
      { $END_IF }
      { $IFDEF pRgb }
      _DevDataX(aNh := VOID(aPar[3]), dst := VOID(pRgb), n:=20);
      { $END_IF }
      { $IFDEF ypWsb }
      _DevDataX(aNh := VOID(aPar[4]), dst := VOID(ypWsb), n := 50);
      { $END_IF }
      { $IFDEF ypTgl }
      _DevDataX(aNh := VOID(aPar[15]), dst := VOID(ypTgl), n := 120);
      { $END_IF }
      { $IFDEF pTla }
      _DevDataX(aNh := VOID(aPar[5]), dst := VOID(ypTla), n:=20);
      { $END_IF }
      { $IFDEF pZas }
      _DevDataX(aNh := VOID(aPar[6]), dst := VOID(pZas));
      { $END_IF }
      { $IFDEF ypPir }
      _DevDataX(aNh := VOID(aPar[7]), dst := VOID(ypPir));
      { $END_IF }
      { $IFDEF ypHEt }
      _DevDataX(aNh := VOID(aPar[9]), dst := VOID(ypHet), n := 20);
      { $END_IF }
      { $IFDEF ypScn }
      _DevDataX(aNh := VOID(aPar[10]), dst := VOID(ypScn), n := 20);
      { $END_IF }
      { $IFDEF ypRol }
      _DevDataX(aNh := VOID(aPar[12]), dst := VOID(ypRol), n:=100);
      { $END_IF }
      { $IFDEF ypGat }
      _DevDataX(aNh := VOID(aPar[13]), dst := VOID(ypGat));
      { $END_IF }
      { $IFDEF yCox }
      _DevDataX(aNh := VOID(aCfg[41]), dst := VOID(yCox), n :=10);
      { $END_IF }
      { $IFDEF pDls }
      _DevDataX(aNh := VOID(aPar[16]), dst := VOID(pDLs), n := 200);
      { $END_IF }

// WRK
      { $IFDEF yCaW }
//         memset(val := 0, length := aSys.sCaW, dest := VOID( mRam[aSys.aCaW1] ));
         MemcpyEx(length :=  aSys.sCaW  , source := void( mRam[aSys.aCaW1] ), dest := VOID(yCaW));
      { $END_IF }
      { $IFDEF yRoW }
         MemcpyEx(length :=  MIN(10,aSys.sRoW/SIZEOF(NH_WRK_ROM))  , source := void( mRam[aSys.aRoW1] ), dest := VOID(yRoW));
      { $END_IF }
      { $IFDEF yZoW }
         MemcpyEx(length :=  MIN( 7,aSys.sRoW/SIZEOF(NH_WRK_ROM))  , source := void( mRam[aSys.aZoW1] ), dest := VOID(yZoW));
      { $END_IF }

      { $IFDEF yIdx }
         memset(val := 0, length := 30 * SIZEOF(NH_IDX), dest := VOID(yIdx));
         MemcpyEx(length :=  MIN(30,USINT_TO_UDINT(aWeb.M[1].ixb[0].idx + aWeb.M[1].ixb[1].idx)) * SIZEOF(NH_IDX)  , source := void( mRam[aSys.vIx1] ), dest := VOID(yIdx));
      { $END_IF }

   END_FUNCTION

{ $ ELSE }
   VAR_GLOBAL                                            // len pre ladenie
      _NhWrk      {HIDDEN} : BOOL := false;
   END_VAR
{ $END_IF }

(* ---- cust.st ---- *)
                       FUNCTION _Nh_CUST_RESTART  {HIDDEN} : BOOL

END_FUNCTION

VAR_GLOBAL
//	_rom_		{HIDDEN}				AT mObr	: USINT;		// pouzita len pre mapovanie rom koli exportu
	_rom_		{HIDDEN}				:BOOL;
   ROM_101	{HIDDEN}{PUBLIC} 	AT _rom_;            //Pepo;1
   ROM_102	{HIDDEN}{PUBLIC} 	AT _rom_;            //Spalna;1
   ROM_000	{HIDDEN}{PUBLIC} 	AT _rom_;            //System;0
   ROM_X02  {HIDDEN}{PUBLIC} 	AT _rom_; 				//Balkon;2
   ROM_X01  {HIDDEN}{PUBLIC} 	AT _rom_;            //Vonku;2

	GAT_X01			{PUBLIC} : BOOL;                 //Garáž-L;X01
	GAT_X02			{PUBLIC} : BOOL;                 //Garáž-P;X01
	GAT_X04_1		{PUBLIC} : BOOL;                 //Brána;X01
	GAT_X04_Y		{PUBLIC} : BOOL;                 //brana-zatvorit;X01
	GAT_X05_2		{PUBLIC} : BOOL;                 //Bránièka;X01
	GAT_X03_3		{PUBLIC} : BOOL;                 //Vstup.dvere;X01

	ZAS_000			{PUBLIC} : BOOL;                 //Zásuvka ON/OFF;102
	ZAS_001_1		{PUBLIC} : BOOL;                 //Zásuvka-Lampa;102
	ZAS_002_2		{PUBLIC} : BOOL;                 //Stykaè-ON;102
	ZAS_003_3		{PUBLIC} : BOOL;                 //Stykaè-OFF;102
	ZAS_004_4		{PUBLIC} : BOOL;                 //Zásuvka-ohrievaè;102
	ZAS_005_5		{PUBLIC} : BOOL;                 //Zásuvka-ventilátor;102
	ZAS_006_6      {PUBLIC} : BOOL;                 //Nabijacia stanica;102
	ZAS_009_9      {PUBLIC} : BOOL;                 //HW-Reset;102

END_VAR

(*
VAR_GLOBAL CONSTANT

   _NewDbx  : BOOL := 0;      // natvrdo sa po restarte vytvaraju vsetky nove dat1
//   _GoExp   : BOOL := 1;      // ide sa do exportu = exportuju sa vety CFG a postupuje sa podla ActHWA

	_NhIpWebPush	: string [16]		:='192.168.9.175';
	{$IFDEF __NH_DALI}
		_Nh_DALI_MA	{HIDDEN} : USINT	:=  2;			 									// pocet samostatnych sad vazieb aVaz[_Nh_VIO]
   {$END_IF}
	{ $IFDEF __NH_METEO_IQWS_4000 }
		_NhipIQWS       	 : string [16]		:='192.168.43.100'; 	//IP adresa anemometru IQWS 4000
	{ $END_IF}

 	_Nh_MSG	{HIDDEN} : USINT			:= 1;				// celkovy pocet formularov

	_Nh_MSG_RCV	: ARRAY[1..1] OF STRING[80] := [
	'f7ab034164f9378b1f2b65fd0554f912c0e2272f43a9d2e6fa25d377c65031cf'   	// moje
//	'.af2f65949afbc152c0d77eebb9aaf5d5cca5930cdc3057f52635c8301106c8b6',    	// Marek
//	'db9e76ae6a095bb2450409752c48b065f3cea3a5caf2f47401a3ece10ee6ea8e',	   // mamka
//	'87e08ab8c8c05dd0732292b70bf14649ed2e69ba4d363177a7d19c26196cfc21'      // Zuzka M.
	];

(*
	_Nh_MSG_NBR	{HIDDEN} : USINT			:= 1;											// celkovy pocet formularov
	_Nh_MSG_TOKEN	: ARRAY[1..3] OF STRING[80] := [
	'f7ab034164f9378b1f2b65fd0554f912c0e2272f43a9d2e6fa25d377c65031cf',  	// moje
	'db9e76ae6a095bb2450409752c48b065f3cea3a5caf2f47401a3ece10ee6ea8e',	   // mamka
	'A'
//	'db9e76ae6a095bb2450409752c48b065f3cea3a5caf2f47401a3ece10ee6ea8e',	   // mamka
//	'87e08ab8c8c05dd0732292b70bf14649ed2e69ba4d363177a7d19c26196cfc21'      // Zuzka M.
	];

END_VAR
*)
(*
VAR_GLOBAL
	rr					: BOOl;
   ROM_101        {PUBLIC} AT rr;                 //Pepo;1
   ROM_102        {PUBLIC} AT rr;                 //Spalna;1
   ROM_000         {PUBLIC} AT rr;                //System;0
   ROM_X02       {PUBLIC} AT rr;                 //Balkon;2
   ROM_X01       {PUBLIC} AT rr;                 //Vonku;2

	GAT_X01			{PUBLIC} : BOOL;                 //Garáž-L;X01
	GAT_X02			{PUBLIC} : BOOL;                 //Garáž-P;X01
	GAT_X04_1		{PUBLIC} : BOOL;                 //Brána;X01
	GAT_X04_Y		{PUBLIC} : BOOL;                 //brana-zatvorit;X01
	GAT_X05_2		{PUBLIC} : BOOL;                 //Bránièka;X01
	GAT_X03_3		{PUBLIC} : BOOL;                 //Vstup.dvere;X01

	ZAS_000			{PUBLIC} : BOOL;                 //Zásuvka ON/OFF;102
	ZAS_001_1		{PUBLIC} : BOOL;                 //Zásuvka-Lampa;102
	ZAS_002_2		{PUBLIC} : BOOL;                 //Stykaè-ON;102
	ZAS_003_3		{PUBLIC} : BOOL;                 //Stykaè-OFF;102
	ZAS_004_4		{PUBLIC} : BOOL;                 //Zásuvka-ohrievaè;102
	ZAS_005_5		{PUBLIC} : BOOL;                 //Zásuvka-ventilátor;102
	ZAS_006_6      {PUBLIC} : BOOL;                 //Nabijacia stanica;102
	ZAS_009_9      {PUBLIC} : BOOL;                 //HW-Reset;102
END_VAR
*)
